# EPICS autosave request: hexmapApp/Db/NDHexMap_settings.req
$(P)$(R)Type
$(P)$(R)NewSizeX
$(P)$(R)NewSizeY
$(P)$(R)HexPitch
file "NDPluginBase_settings.req", P=$(P), R=$(R)
